// TwinCAT 3 PLC project Untitled1
// ProgramVersion: 3.1.4023.0
// libraries:
//   Tc2_MC2, * (Beckhoff Automation GmbH)
//   Tc2_Standard, * (Beckhoff Automation GmbH)
//   Tc2_System, * (Beckhoff Automation GmbH)
//   Tc3_Module, * (Beckhoff Automation GmbH)
// project tree:
//   DUTs/ Conv1.TcDUT, Conv2.TcDUT, StructAxis.TcDUT
//   GVLs/ IO.TcGVL
//   / PlcTask.TcTTO
//   POUs/ MAIN.TcPOU, StepperProg.TcPOU
// real-time tasks:
//   TASK PlcTask: cycle T#10ms, priority 20, ADS port 350
// motion (NC):
//   TASK NC-Task 1 SAF: cycle T#2ms, priority 4, ADS port 501
//   TASK NC-Task 1 SVB: cycle T#10ms, priority 8, ADS port 511
//   AXIS Axis 1 (id 1)
//     General: UnitName=°
//     Dynamic: DelayTime=0.008
//     Velo: Maximum=3300
//     OtherSettings: AllowMotionCmdToSlave=true
//     encoder EncType=4
//       EncPara: ScaleFactorNumerator=0.028125, MaxCount=#x0000ffff
//         Inc: RefSoftSyncMask=#x0000ffff
//         TimeComp: TimeCompMode=1, EncDelayCycles=4
//     drive DrvType=24
//       Analog: VeloReferenz=3600, TorqueSetpointScale=10, ScaleFactorActTorque=0.1
//       TimeComp: TaskDelayCycles=1
//     controller CtrType=1
//       CtrPara: PriorControlFactor=1
//         Observer: BandWidth=20
//   AXIS Axis 2 (id 2)
//     General: UnitName=°
//     Dynamic: Acceleration=19380, Deceleration=19380, Jerk=38760, DelayTime=0.008
//     Velo: RefSearch=291.78, RefSync=291.78, SlowManual=1458.9, FastManual=8753.4, Fast=29178, Maximum=9690
//     OtherSettings: AllowMotionCmdToSlave=true
//     encoder EncType=19
//       EncPara: ScaleFactorNumerator=360, ScaleFactorDenominator=1048576, MaxCount=#xffffffff
//         TimeComp: TimeCompMode=1, EncDelayCycles=4
//     drive DrvType=16
//       DrvPara: MaxCount=#xffffffff, DriveControlDWord=#x00020000
//         Analog: VeloReferenz=10659, VeloScale=32, TorqueSetpointScale=10, ScaleFactorActTorque=0.1
//         TimeComp: TaskDelayCycles=1
//     controller CtrType=1
//       CtrPara: PriorControlFactor=1
//         Observer: BandWidth=20
// I/O:
//   DEVICE Device 1 (EtherCAT), AmsNetId 5.78.138.248.2.1
//     Term 1 (EK1200) [EK1200-5000 EtherCAT Power supply (2A E-Bus)]
//       Term 2 (EL1014) [EL1014 4Ch. Dig. Input 24V, 10µs]
//       Term 3 (EL2014) [EL2014 4Ch. Dig. Output 24V, 0,5A, Diagnostic]
//       Term 4 (EL6910) [EL6910, TwinSAFE PLC]
//       Term 5 (EL1904) [EL1904, 4 Ch. Safety Input 24V, TwinSAFE]
//         modules: Module 1 (FSOES)
//       Term 6 (EL3102) [EL3102 2Ch. Ana. Input +/-10V, Diff.]
//       Term 7 (EL4102) [EL4102 2Ch. Ana. Output  0-10V, 16bit]
//       Term 8 (EL9512) [EL9512 Power supply terminal 12V]
//       Term 9 (EK1122) [EK1122 2 port EtherCAT junction]
//       Term 10 (EK1110) [EK1110 EtherCAT extension]
//     Term 11 (EK1101) [EK1101 EtherCAT Coupler (2A E-Bus, ID switch)]
//       Term 12 (EL1809) [EL1809 16Ch. Dig. Input 24V, 3ms]
//       Term 13 (EL2809) [EL2809 16Ch. Dig. Output 24V, 0.5A]
//       Term 14 (EL2904) [EL2904, 4 Ch. Safety Output 24V, 0.5A, TwinSAFE]
//         modules: Module 1 (FSOES), Module 2 (DO)
//       Term 15 (EL6021) [EL6021 Interface (RS422/485)]
//       Term 16 (EL9110) [EL9110 Power Supplier with LED (24V, Diagnostics)]
//       Term 17 (EL7031) [EL7031 1Ch. Stepper motor output stage (24V, 1.5A)]
//       Term 18 (EL7201-9014) [EL7201-9014 1Ch. MDP742 Servo motor output stage with OCT (50V, 2.8A RMS) and STO input]
//       Term 19 (EL9011) [EL9011 End Terminal]
// variable links:
//   NC-Task 1 SAF/Axes/Axis 1 <-> Device 1 (EtherCAT)/Term 11 (EK1101)/Term 17 (EL7031)
//     Drive/Inputs/In/nState1 @bit 3 <-> STM Status/Status/Error
//     Drive/Inputs/In/nState1 @bit 5 <-> STM Status/Status/Moving negative
//     Drive/Inputs/In/nState1 @bit 4 <-> STM Status/Status/Moving positive
//     Drive/Inputs/In/nState1 @bit 1 <-> STM Status/Status/Ready
//     Drive/Inputs/In/nState1 <-> STM Status/Status/Ready to enable
//     Drive/Inputs/In/nState1 @bit 6 <-> STM Status/Status/Torque reduced
//     Drive/Inputs/In/nState1 @bit 2 <-> STM Status/Status/Warning
//     Drive/Inputs/In/nState2 @bit 3 <-> STM Status/Status/Digital input 1
//     Drive/Inputs/In/nState2 @bit 4 <-> STM Status/Status/Digital input 2
//     Drive/Inputs/In/nState2 @bit 5 <-> STM Status/Status/Sync error
//     Drive/Inputs/In/nState2 @bit 7 <-> STM Status/Status/TxPDO Toggle
//     Drive/Inputs/In/nState4 @bit 1 <-> WcState/InputToggle
//     Drive/Inputs/In/nState4 <-> WcState/WcState
//     Drive/Outputs/Out/nCtrl1 <-> STM Control/Control/Enable
//     Drive/Outputs/Out/nCtrl1 @bit 2 <-> STM Control/Control/Reduce torque
//     Drive/Outputs/Out/nCtrl1 @bit 1 <-> STM Control/Control/Reset
//     Drive/Outputs/Out/nDataOut2[0] <-> STM Velocity/Velocity
//     Enc/Inputs/In/nDataIn1[0] <-> ENC Status compact/Counter value
//     Enc/Inputs/In/nDataIn2[0] <-> ENC Status compact/Latch value
//     Enc/Inputs/In/nState1 @bit 4 <-> ENC Status compact/Status/Counter overflow
//     Enc/Inputs/In/nState1 @bit 3 <-> ENC Status compact/Status/Counter underflow
//     Enc/Inputs/In/nState1 @bit 1 <-> ENC Status compact/Status/Latch extern valid
//     Enc/Inputs/In/nState1 @bit 2 <-> ENC Status compact/Status/Set counter done
//     Enc/Inputs/In/nState2 @bit 4 <-> ENC Status compact/Status/Status of extern latch
//     Enc/Inputs/In/nState2 @bit 5 <-> ENC Status compact/Status/Sync error
//     Enc/Inputs/In/nState2 @bit 7 <-> ENC Status compact/Status/TxPDO Toggle
//     Enc/Inputs/In/nState4 @bit 1 <-> WcState/InputToggle
//     Enc/Inputs/In/nState4 <-> WcState/WcState
//     Enc/Outputs/Out/nCtrl1 @bit 3 <-> ENC Control compact/Control/Enable latch extern on negative edge
//     Enc/Outputs/Out/nCtrl1 @bit 1 <-> ENC Control compact/Control/Enable latch extern on positive edge
//     Enc/Outputs/Out/nCtrl1 @bit 2 <-> ENC Control compact/Control/Set counter
//     Enc/Outputs/Out/nDataOut1[0] <-> ENC Control compact/Set counter value
//   NC-Task 1 SAF/Axes/Axis 2 <-> Device 1 (EtherCAT)/Term 11 (EK1101)/Term 18 (EL7201-9014)
//     Drive/Inputs/In/nDcOutputTime <-> InfoData/DcOutputShift
//     Drive/Inputs/In/nState1 <-> DRV Statusword/Statusword
//     Drive/Inputs/In/nState2 <-> DRV Statusword/Statusword @bit 8
//     Drive/Inputs/In/nState4 @bit 1 <-> WcState/InputToggle
//     Drive/Inputs/In/nState4 <-> WcState/WcState
//     Drive/Outputs/Out/nCtrl1 <-> DRV Controlword/Controlword
//     Drive/Outputs/Out/nCtrl2 <-> DRV Controlword/Controlword @bit 8
//     Drive/Outputs/Out/nDataOut2 <-> DRV Target velocity/Target velocity
//     Enc/Inputs/In/nDataIn1 <-> FB Position/Position
//     Enc/Inputs/In/nDcInputTime <-> InfoData/DcInputShift
//     Enc/Inputs/In/nState4 @bit 1 <-> WcState/InputToggle
//     Enc/Inputs/In/nState4 <-> WcState/WcState
//   Untitled1/Untitled1 Instance <-> Device 1 (EtherCAT)/Term 1 (EK1200)/Term 2 (EL1014)
//     PlcTask Inputs/IO.bSwitch{1..4} <-> Channel {1..4}/Input  (4 links)
//   Untitled1/Untitled1 Instance <-> Device 1 (EtherCAT)/Term 1 (EK1200)/Term 3 (EL2014)
//     PlcTask Outputs/IO.bLed{1..4} <-> DIG Outputs/Channel {1..4}/Output  (4 links)
//   Untitled1/Untitled1 Instance <-> NC-Task 1 SAF/Axes/Axis 1
//     PlcTask Inputs/MAIN.StepperAxis.NcToPlc <-> Outputs/ToPlc
//     PlcTask Outputs/MAIN.StepperAxis.PlcToNc <-> Inputs/FromPlc
//   Untitled1/Untitled1 Instance <-> NC-Task 1 SAF/Axes/Axis 2
//     PlcTask Inputs/MAIN.ServoAxis.NcToPlc <-> Outputs/ToPlc
//     PlcTask Outputs/MAIN.ServoAxis.PlcToNc <-> Inputs/FromPlc

CONFIGURATION Untitled1
    RESOURCE PLC ON TwinCAT3
        TASK PlcTask(INTERVAL := T#10ms, PRIORITY := 20);
        PROGRAM MAIN WITH PlcTask : MAIN;
    END_RESOURCE
END_CONFIGURATION

// ---- DUTs/Conv1.TcDUT
{attribute 'qualified_only'}
{attribute 'strict'}
TYPE Conv1 :
(
	Init :=0,
	Enable,
	Conv1ON,
	Conv1OFF,
	Conv1Stop,
	tim1,
	MoveForwards,
	Error,
	Reset
);
END_TYPE

// ---- DUTs/Conv2.TcDUT
{attribute 'qualified_only'}
{attribute 'strict'}
TYPE Conv2 :
(
	Init :=0,
	Enable,
	Conv2ON,
	Conv2OFF,
	Conv2Stop,
	MoveForwards,
	Error,
	Reset
);
END_TYPE

// ---- DUTs/StructAxis.TcDUT
TYPE StructAxis :
STRUCT
	Power : MC_Power;
	Reset : MC_Reset;
	MoveAbs : MC_MoveAbsolute;
	MoveRel : MC_MoveRelative;
	halt : MC_Halt;
	MoveVel : MC_MoveVelocity;
	McStop : MC_Stop;
END_STRUCT
END_TYPE

// ---- GVLs/IO.TcGVL
{attribute 'qualified_only'}
VAR_GLOBAL
		// Digital Input
		bSwitch1 AT %I* : BOOL;
		bSwitch2 AT %I* : BOOL;
		bSwitch3 AT %I* : BOOL;
		bSwitch4 AT %I* : BOOL;
		
	//Digital Output
		bLed1 AT %Q* : BOOL;
		bLed2 AT %Q* : BOOL;
		bLed3 AT %Q* : BOOL;
		bLed4 AT %Q* : BOOL;
		
	//Analog Input
		nResistor1 AT %I* : INT;
		nResistor2 AT %I* : INT;
		
	//Analog Output
		nVoltmeter1 AT %Q* : INT;
		nVoltmeter2 AT %Q* : INT;
END_VAR

// ---- POUs/MAIN.TcPOU
PROGRAM MAIN
VAR
	Servo : StructAxis;		//CONV 1
	Stepper : StructAxis;	//CONV2
	
	ServoAxis : AXIS_REF;
	StepperAxis : AXIS_REF;
	oState : Conv2;
	iState : Conv1;
	
	tim1 : TON;
END_VAR

ACT_Move();
ACT_Power();
ACT_Reset();
ACT_Stop();

CASE iState OF 
	Conv1.Init: 						// setting intial position of Conv1
		tim1(IN:=FALSE);
		servo.MoveVel.Execute :=FALSE;  
		servo.Reset.Execute :=FALSE;
		
		iState := Conv1.Enable; // move to next step(enabling servo motor)
		
	Conv1.Enable:					// Power up the Servo motor
		servo.Power.Enable := TRUE;
		servo.Power.Enable_Positive := TRUE;
	    servo.Power.Enable_Negative := TRUE;
		
		IF servo.Power.Status THEN
			iState := Conv1.Conv1ON;
 		ELSIF servo.Power.Error THEN
			iState := Conv1.Error;
		END_IF
		
	Conv1.Conv1ON:
		IF IO.bSwitch1 THEN						// Start button pressed
			IO.bLed1 := TRUE;					// show logic works
			iState := Conv1.MoveForwards;// Conv1 move forward
		
		END_IF
	Conv1.MoveForwards:
		tim1(IN:=FALSE);
	
		Servo.MoveVel.Execute := TRUE;
		Servo.MoveVel.Velocity := 100;
	
		IF IO.bSwitch2 THEN					// if "Box" is detected on Conv1
			IO.bLed2 := TRUE;
			servo.MoveVel.Execute := FALSE;
			iState := Conv1.Conv1Stop; 		// Conv1 Stop
		IF IO.bSwitch2 AND IO.bSwitch4 THEN
			iState := Conv1.tim1;
		END_IF
		END_IF
		
	Conv1.tim1:
			tim1(IN := TRUE,PT := T#5S);
			IF tim1.Q THEN
				iState := Conv1.MoveForwards;
			END_IF
			
	Conv1.Conv1Stop:
		Servo.McStop.Execute := TRUE;
				
		IF Servo.McStop.Done THEN
			Servo.McStop.Execute := FALSE;
			iState := Conv1.MoveForwards;
		END_IF
		
	IF servo.MoveVel.Error OR servo.MoveVel.CommandAborted THEN // if error or sudden estop initiated
			iState := Conv1.Error;
			stepper.MoveVel.Execute :=FALSE;
			
		END_IF
		
	Conv1.Error:													// if error, stop n reset
		IF StepperAxis.Status.Error  THEN
			iState := Conv1.Reset;
		ELSE
			iState := Conv1.Init;
		END_IF
		
	Conv1.Reset:
		Servo.Reset.Execute := TRUE;
		
		
		IF  servo.Reset.Done THEN
			iState := Conv1.Init;
		ELSIF servo.Reset.Error THEN
			iState := Conv1.Error;
		END_IF
	
	

END_CASE
//////////////////////////////////////////////////////////////////////////////////////////////////////////////////////////////////////////////////////////////////////////////////////////////////////////////
			CASE oState OF 
				Conv2.Init: 						// setting intial position of Conv2
					Stepper.MoveVel.Execute :=FALSE;  
					stepper.Reset.Execute :=FALSE;
					Servo.McStop.Execute := FALSE;
					oState := Conv2.Enable; // move to next step(enabling stepper motor)
					
				Conv2.Enable:					// Power up the stepper motor
					stepper.Power.Enable := TRUE; 
					stepper.Power.Enable_Positive := TRUE; // Ensure it is able to turn positive and negative
					stepper.Power.Enable_Negative := TRUE;
				   
					
					IF Stepper.Power.Status THEN
						oState := Conv2.Conv2ON;
			 		ELSIF Stepper.Power.Error THEN
						oState := Conv2.Error;
					END_IF
					
				Conv2.Conv2ON:
					IF IO.bSwitch1 THEN						// Start button pressed
						IO.bLed1 := TRUE;					// show logic works
						oState := Conv2.MoveForwards;		// Conv2 move forward
					ELSE IO.bLed1 := FALSE;
					END_IF
					
				Conv2.MoveForwards:
				
						stepper.MoveVel.Execute := TRUE;
						stepper.MoveVel.Velocity := 100;
					
					IF IO.bSwitch3 THEN					// if "Object" is detected on Conv2
						IO.bLed3 := TRUE;
						Stepper.MoveVel.Execute := FALSE;
						oState := Conv2.Conv2Stop;	 	// Conv2 Stop
					END_IF
					
				Conv2.Conv2Stop:
					stepper.McStop.Execute := TRUE;
							
					IF NOT IO.bSwitch3 THEN
						Stepper.McStop.Execute := FALSE;
						oState := Conv2.MoveForwards;
					END_IF
					
				IF Stepper.MoveVel.Error OR Stepper.MoveVel.CommandAborted THEN // if error or sudden estop initiated
						oState := Conv2.Error;
						stepper.MoveVel.Execute :=FALSE;
						
					END_IF
					
				Conv2.Error:													// if error, stop n reset
					IF StepperAxis.Status.Error  THEN
						oState := Conv2.Reset;
					ELSE
						oState := Conv2.Init;
					END_IF
					
				Conv2.Reset:
					Stepper.Reset.Execute := TRUE;
					
					IF  Stepper.Reset.Done THEN
						oState := Conv2.Init;
					ELSIF Stepper.Reset.Error THEN
						oState := Conv2.Error;
					END_IF
				
			END_CASE

ACTION ACT_Move:
Servo.MoveVel(Axis := ServoAxis);
	
Stepper.MoveVel( Axis := StepperAxis);
END_ACTION

ACTION ACT_Power:
Servo.Power( Axis := ServoAxis);

Stepper.Power( Axis := StepperAxis);
END_ACTION

ACTION ACT_Reset:
Servo.Reset( Axis := ServoAxis);

Stepper.Reset( Axis := StepperAxis);
END_ACTION

ACTION ACT_Stop:
Servo.McStop(Axis := ServoAxis);
	
Stepper.McStop( Axis := StepperAxis);
END_ACTION

END_PROGRAM

// ---- POUs/StepperProg.TcPOU
PROGRAM StepperProg
VAR
		Servo : StructAxis;		//CONV 1
	Stepper : StructAxis;	//CONV2
	
	ServoAxis : AXIS_REF;
	StepperAxis : AXIS_REF;
	oState : Conv2;
END_VAR

CASE oState OF 
	Conv2.Init: 						// setting intial position of Conv2
		Stepper.MoveVel.Execute :=FALSE;  
		stepper.Reset.Execute :=FALSE;
		Servo.McStop.Execute := FALSE;
		oState := Conv2.Enable; // move to next step(enabling servo motor)
		
	Conv2.Enable:					// Power up the stepper motor
		stepper.Power.Enable := TRUE; 
		stepper.Power.Enable_Positive := TRUE; // Ensure it is able to turn positive and negative
		stepper.Power.Enable_Negative := TRUE;
	   
		
		IF servo.Power.Status THEN
			oState := Conv2.Conv2ON;
 		ELSIF servo.Power.Error THEN
			oState := Conv2.Error;
		END_IF
		
	Conv2.Conv2ON:
		IF IO.bSwitch1 THEN						// Start button pressed
			IO.bLed1 := TRUE;					// show logic works
			oState := Conv2.MoveForwards;// Conv1 move forward
		END_IF
		
	Conv2.MoveForwards:
	
		//stepper.MoveAbs.Position := 3600;
		//stepper.MoveAbs.Velocity := 50; 
	
			stepper.MoveVel.Execute := TRUE;
			stepper.MoveVel.Velocity := 100;
		
		//stepper.MoveAbs.Execute :=TRUE; 
	
		IF IO.bSwitch3 THEN					// if "Object" is detected on Conv2
			IO.bLed3 := TRUE;
			//iState := Conv1.Conv1OFF;
			servo.MoveVel.Execute := FALSE;
			oState := Conv2.Conv2Stop; // Conv2 Stop
		END_IF
		
(*		IF IO.bSwitch3 THEN					// if "object" is detected on Conv2
			iState := E_MoveState.Conv2OFF; // Conv2 stop
		END_IF
*)	
	//Conv1.Conv1OFF:					// Stop Servo(Conv1)
	//	servo.MoveVel.Execute := FALSE;
	//	iState := Conv1.Conv1Stop;
		
	Conv2.Conv2Stop:
		Servo.McStop.Execute := TRUE;
				
		IF Servo.McStop.Done THEN
			oState := Conv2.Init;
		END_IF
		

(*	Conv2.Conv2OFF:					// Stop Stepper(Conv2)
		Stepper.MoveAbs.Execute :=FALSE;
		IF NOT IO.bSwitch3 AND IO.bSwitch1 THEN
			iState := E_MoveState.Conv2ON;
		END_IF
*)		
(*	Conv2.Conv2ON:					//On Stepper(Conv2)
		stepper.MoveAbs.Position := 3600;
		stepper.MoveAbs.Velocity := 50; 
		stepper.MoveAbs.Execute :=TRUE;
*)		
	IF servo.MoveVel.Error OR servo.MoveVel.CommandAborted THEN // if error or sudden estop initiated
			oState := Conv2.Error;
			stepper.MoveVel.Execute :=FALSE;
			
		END_IF
		
	Conv1.Error:													// if error, stop n reset
		IF StepperAxis.Status.Error  THEN
			oState := Conv2.Reset;
		ELSE
			oState := Conv2.Init;
		END_IF
		
	Conv1.Reset:
		Stepper.Reset.Execute := TRUE;
		
		
		IF  servo.Reset.Done THEN
			oState := Conv2.Init;
		ELSIF servo.Reset.Error THEN
			oState := Conv2.Error;
		END_IF
	
	

END_CASE

END_PROGRAM
